# B&R Automation Studio project WRAPPER_CTRL
Automation Studio 4.9.6.42 SP; technology packages: mapp 1.63.0

## Configuration Errepi_P00936

CPU X20CP1301, AutomationRuntime O4.34, Build 4.1.2, Vc V4.72.7

### Task classes (Cpu.sw)
```
Cyclic#1 (cycle 8000 us, tolerance 8000 us):
  clock <- clock.prg
  Varie <- Varie.prg
  Program <- (binary)
Cyclic#2:
  main <- main.prg
Binaries: udbdef, TCData, sysconf, Role, User, iomap, ashwd, asfw, arconfig, ashwac
Libraries: FileIO, runtime, astime, asieccon, standard
```

### Hardware
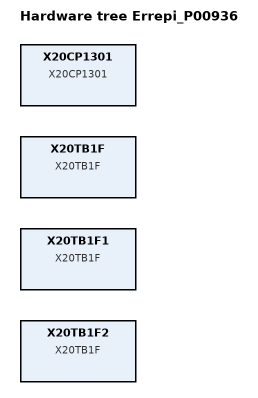
```
X20CP1301 : X20CP1301 v1.7.0.0  [X1 -> X1.SL; X2 -> X2.SL; X3 -> X3.SL]
  Module X1 (Type=X1, Virtual=true, Version=1.7.0.0)
    Connection (Connector=SS1, TargetModule=X20TB1F, TargetConnector=SS)
    Connection (Connector=SL, TargetModule=X20CP1301, TargetConnector=X1)
  Module X2 (Type=X2, Virtual=true, Version=1.7.0.0)
    Connection (Connector=SS1, TargetModule=X20TB1F1, TargetConnector=SS)
    Connection (Connector=SL, TargetModule=X20CP1301, TargetConnector=X2)
  Module X3 (Type=X3, Virtual=true, Version=1.7.0.0)
    Connection (Connector=SS1, TargetModule=X20TB1F2, TargetConnector=SS)
    Connection (Connector=SL, TargetModule=X20CP1301, TargetConnector=X3)
  Connector IF2:
    ActivateDevice = 1
    HostName = p00936
    Mode = Manual
    InternetAddress = 192.168.49.7
    SubnetMask = 255.255.255.0
    Vnc1
    VncVcObjectName1 = Visu
    VncKeyMappingFile1 = VC\PS2-Keyboard.dis
    VncAuthentication1 = 1
    VncPasswordViewOnly1 = errepi
    VncPasswordViewControl1 = promass
    ActivateSnmp = 2
  ConfigurationID = ERREPI_P00936
  ConfigVersion = 2022.5.1
  PermanentPvSize = 35
  RemanentGlobalPvSize = 45
  EnableUsbRemoteInstall = 1
  EnableCfRemoteInstall = 1
  RebootReset = 1
  Connections = 10
  TimerDeviceType = EPLX2X
  TimerDevice = X20CP1301.IF6
  TaskClassIdleTime = 8000
  Cyclic1Duration = 8000
  Cyclic1Tolerance = 8000
  Cyclic3Duration = 48000
  Cyclic3Tolerance = 48000
  Cyclic8Duration = 8000
  FileDevice1
  FileDeviceName1 = HD
  FileDevicePath1 = D:\RECIPES\
  FileDevice2
  FileDeviceName2 = CF
  FileDevicePath2 = D:\
  FileDevice3
  FileDeviceName3 = LOG
  FileDevicePath3 = D:\LOG\
  ActivateSntp = 1
  SntpcServAddr1 = 192.168.49.1
  SntpcServAddr2 = 8.8.8.8
  InternetFileSystemUsername = promass
  InternetFileSystemPassword = promass
  EthernetHostName = p00936
  EthernetDefaultGateway = 192.168.49.1
  FtpUser1
  FtpUsername1 = bazzica
  FtpUserPassword1 = fv7Wv821ewKqnMsDSvGQxxKgMMgXs+bZF/2FwIesLr0=  // promass
  FtpUserSalt1 = UDA6md8F
  FTPAccessRight1 = 0
  FTPMSPartition1 = DATA
  FtpUser2
  FtpUsername2 = errepi
  FtpUserPassword2 = knNz1PPTdcY0SkTRJpi6SMuvDsE3Y9gUDrG6vRz9RC4=  // errepi
  FtpUserSalt2 = Ww6eA1cq
  FTPAccessRight2 = 0
  FTPMSPartition2 = DATA
  ActivateOpcUa = 1
  OpcUaInformationModels_PV_Version = 1
X20TB1F : X20TB1F v1.0.0.0
X20TB1F1 : X20TB1F v1.0.0.0
X20TB1F2 : X20TB1F v1.0.0.0
```

### Cpu.per - X20CP1301/Cpu.per
```iecst
VAR_CONFIG
	gMac01LifeCounter AT %MD0; (* *)
	gMac01CounterOffset AT %MD4; (* *)
	gMac02LifeCounter AT %MD8; (* *)
	gMac02CounterOffset AT %MD12; (* *)
	gMac03LifeCounter AT %MD16; (* *)
	gMac03CounterOffset AT %MD20; (* *)
	glb_mac_name AT %M24; (* *)
END_VAR
```

## Configuration Errepi_P00987

CPU X20CP1301, AutomationRuntime O4.34, Build 4.1.2, Vc V4.72.7

### Hardware
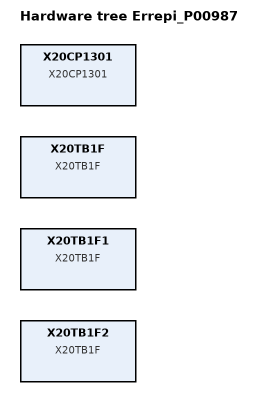
```
X20CP1301 : X20CP1301 v1.7.0.0  [X1 -> X1.SL; X2 -> X2.SL; X3 -> X3.SL]
  Module X1 (Type=X1, Virtual=true, Version=1.7.0.0)
    Connection (Connector=SS1, TargetModule=X20TB1F, TargetConnector=SS)
    Connection (Connector=SL, TargetModule=X20CP1301, TargetConnector=X1)
  Module X2 (Type=X2, Virtual=true, Version=1.7.0.0)
    Connection (Connector=SS1, TargetModule=X20TB1F1, TargetConnector=SS)
    Connection (Connector=SL, TargetModule=X20CP1301, TargetConnector=X2)
  Module X3 (Type=X3, Virtual=true, Version=1.7.0.0)
    Connection (Connector=SS1, TargetModule=X20TB1F2, TargetConnector=SS)
    Connection (Connector=SL, TargetModule=X20CP1301, TargetConnector=X3)
  Connector IF2:
    ActivateDevice = 1
    HostName = p00987
    Mode = Manual
    InternetAddress = 192.168.49.2
    SubnetMask = 255.255.255.0
    Vnc1
    VncVcObjectName1 = Visu
    VncKeyMappingFile1 = VC\PS2-Keyboard.dis
    VncAuthentication1 = 1
    VncPasswordViewOnly1 = errepi  // Password: errepi
    VncPasswordViewControl1 = promass  // Password: promass
    ActivateSnmp = 2
  ConfigurationID = ERREPI_P00987
  ConfigVersion = 2022.5.1
  PermanentPvSize = 35
  RemanentGlobalPvSize = 45
  EnableUsbRemoteInstall = 1
  EnableCfRemoteInstall = 1
  RebootReset = 1
  Connections = 10
  TimerDeviceType = EPLX2X
  TimerDevice = X20CP1301.IF6
  TaskClassIdleTime = 8000
  Cyclic1Duration = 8000
  Cyclic1Tolerance = 8000
  Cyclic3Duration = 48000
  Cyclic3Tolerance = 48000
  Cyclic8Duration = 8000
  FileDevice1
  FileDeviceName1 = HD
  FileDevicePath1 = D:\RECIPES\
  FileDevice2
  FileDeviceName2 = CF
  FileDevicePath2 = D:\
  FileDevice3
  FileDeviceName3 = LOG
  FileDevicePath3 = D:\LOG\
  ActivateSntp = 1
  SntpcServAddr1 = 192.168.49.1
  SntpcServAddr2 = 216.239.35.4
  InternetFileSystemUsername = promass
  InternetFileSystemPassword = promass
  EthernetHostName = p00987
  EthernetDefaultGateway = 192.168.49.1
  FtpUser1
  FtpUsername1 = bazzica
  FtpUserPassword1 = fv7Wv821ewKqnMsDSvGQxxKgMMgXs+bZF/2FwIesLr0=  // promass
  FtpUserSalt1 = UDA6md8F
  FTPAccessRight1 = 0
  FTPMSPartition1 = DATA
  FtpUser2
  FtpUsername2 = errepi
  FtpUserPassword2 = knNz1PPTdcY0SkTRJpi6SMuvDsE3Y9gUDrG6vRz9RC4=  // errepi
  FtpUserSalt2 = Ww6eA1cq
  FTPAccessRight2 = 0
  FTPMSPartition2 = DATA
  ActivateOpcUa = 1
  OpcUaInformationModels_PV_Version = 1
X20TB1F : X20TB1F v1.0.0.0
X20TB1F1 : X20TB1F v1.0.0.0
X20TB1F2 : X20TB1F v1.0.0.0
```

## Configuration SIM

CPU X20CP1382, AutomationRuntime D4.83, Build 4.1.2, Vc V4.72.7

### Hardware
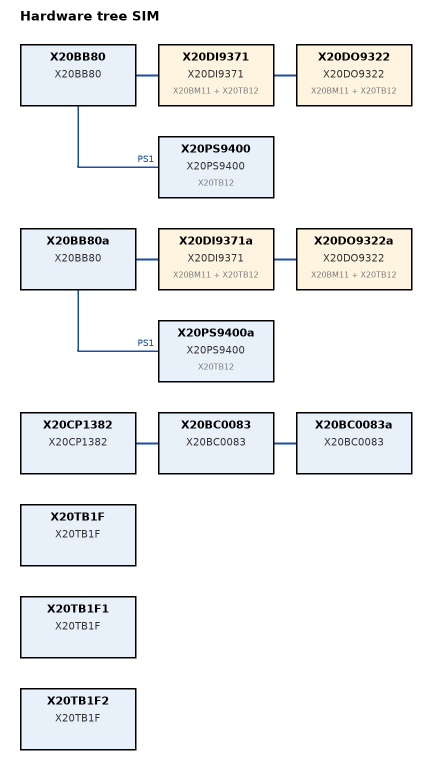
```
X20BB80 : X20BB80 v1.0.2.0
X20BB80a : X20BB80 v1.0.2.0
X20BC0083 : X20BC0083 v2.11.1.0  [PLK1 -> X20CP1382.IF3 (NodeNumber=1) [Cable Type=PowerlinkCable, Length=10, Version=1.0.0.3]; PLK2 -> X20BC0083a.PLK1 (NodeNumber=1) [Cable Type=PowerlinkCable, Length=10, Version=1.0.0.3]; SL -> X20BB80.SL1]
  Supervision = off
X20BC0083a : X20BC0083 v2.11.1.0  [PLK1 -> X20BC0083.PLK2 [Cable Type=PowerlinkCable, Length=10, Version=1.0.0.3]; SL -> X20BB80a.SL1]
  Supervision = off
X20BM11 : X20BM11 v1.0.0.1  [X2X1 -> X20BB80.IF1]
X20BM11a : X20BM11 v1.0.0.1  [X2X1 -> X20BB80a.IF1]
X20BM11b : X20BM11 v1.0.0.1  [X2X1 -> X20BM11.X2X2]
X20BM11c : X20BM11 v1.0.0.1  [X2X1 -> X20BM11a.X2X2]
X20CP1382 : X20CP1382 v1.11.0.0  [X1 -> X1.SL; X2 -> X2.SL; X3 -> X3.SL]
  Module X1 (Type=X1, Virtual=true, Version=1.11.0.0)
    Connection (Connector=SS1, TargetModule=X20TB1F, TargetConnector=SS)
    Connection (Connector=SL, TargetModule=X20CP1382, TargetConnector=X1)
  Module X2 (Type=X2, Virtual=true, Version=1.11.0.0)
    Connection (Connector=SS1, TargetModule=X20TB1F1, TargetConnector=SS)
    Connection (Connector=SL, TargetModule=X20CP1382, TargetConnector=X2)
  Module X3 (Type=X3, Virtual=true, Version=1.11.0.0)
    Connection (Connector=SS1, TargetModule=X20TB1F2, TargetConnector=SS)
    Connection (Connector=SL, TargetModule=X20CP1382, TargetConnector=X3)
  Connector IF2:
    ActivateDevice = 1
    HostName = promass
    Mode = Manual
    InternetAddress = 192.168.3.189  // TURQUEPLAST GIVEN IP
    SubnetMask = 255.255.255.0
    ActivateSnmp = 2
  Connector IF3:
    DNAConfiguration = manual
    CycleTime = 4000
  ConfigurationID = WRAPPER_CTRL_Turqueplast
  SimulationInaNodeNumber = 66
  PermanentPvSize = 1000
  RemanentGlobalPvSize = 20000
  EnableUsbRemoteInstall = 1
  EnableCfRemoteInstall = 1
  RebootReset = 1
  Connections = 10
  TimerDeviceType = EPLX2X
  TimerDevice = X20CP1382.IF3
  TaskClassIdleTime = 8000
  Cyclic1Duration = 8000
  Cyclic1Tolerance = 8000
  Cyclic3Duration = 48000
  Cyclic3Tolerance = 48000
  Cyclic8Duration = 8000
  FileDevice1
  FileDeviceName1 = HD
  FileDevicePath1 = C:\RECIPES\
  FileDevice2
  FileDeviceName2 = CF
  FileDevicePath2 = C:\
  FileDevice3
  FileDeviceName3 = LOG
  FileDevicePath3 = C:\LOG\
  EthernetHostName = promass
  EthernetDefaultGateway = 192.168.3.1
  FtpUser1
  FtpUsername1 = bazzica
  FtpUserPassword1 = VS/6Mr2ZWUxRpzYAgWdC7qPbhzWXz9kZH9v1k0AYU+w=
  FtpUserSalt1 = L4/axyh9
  FTPAccessRight1 = 0
  FTPdevice1 = ALL
  FtpUser2
  FtpUsername2 = turque
  FtpUserPassword2 = NA1x5qBXXFgCR/DJGfRfa8Sh4PrFzhFnpgUflhtmUyQ=
  FtpUserSalt2 = yY9t/zs3
  FTPdevice2 = ALL
X20DI9371 : X20DI9371 v1.1.0.0  [SS1 -> X20TB12b.SS; SL -> X20BM11.SL1]
  Supervision = off
X20DI9371a : X20DI9371 v1.1.0.0  [SS1 -> X20TB12c.SS; SL -> X20BM11a.SL1]
  Supervision = off
X20DO9322 : X20DO9322 v1.3.0.0  [SS1 -> X20TB12d.SS; SL -> X20BM11b.SL1]
  Supervision = off
X20DO9322a : X20DO9322 v1.3.0.0  [SS1 -> X20TB12e.SS; SL -> X20BM11c.SL1]
  Supervision = off
X20PS9400 : X20PS9400 v1.4.0.0  [SS1 -> X20TB12.SS; PS -> X20BB80.PS1]
  Supervision = off
X20PS9400a : X20PS9400 v1.4.0.0  [SS1 -> X20TB12a.SS; PS -> X20BB80a.PS1]
  Supervision = off
X20TB12 : X20TB12 v1.0.0.0
X20TB12a : X20TB12 v1.0.0.0
X20TB12b : X20TB12 v1.0.0.0
X20TB12c : X20TB12 v1.0.0.0
X20TB12d : X20TB12 v1.0.0.0
X20TB12e : X20TB12 v1.0.0.0
X20TB1F : X20TB1F v1.0.0.0
X20TB1F1 : X20TB1F v1.0.0.0
X20TB1F2 : X20TB1F v1.0.0.0
```

### IoMap.iom - X20CP1382/IoMap.iom
```iecst
VAR_CONFIG
	::gPWL02_ok AT %IX."X20BC0083a".ModuleOk;
	::gPWL01_ok AT %IX."X20BC0083".ModuleOk;
END_VAR
```

## Configuration Turqueplast

CPU X20CP1382, AutomationRuntime D4.83, Build 4.1.2, Vc V4.72.7

### Task classes (Cpu.sw)
```
Cyclic#1 (cycle 8000 us, tolerance 8000 us):
  clock <- LOGIC.clock.prg
  Varie <- VARIOUS.Varie.prg
  Program <- (binary)
Cyclic#2:
  main <- LOGIC.main.prg
Binaries: udbdef, TCData, sysconf, Role, User, iomap, ashwd, asfw, arconfig, ashwac
Libraries: FileIO, runtime, astime, asieccon, standard
```

### Hardware
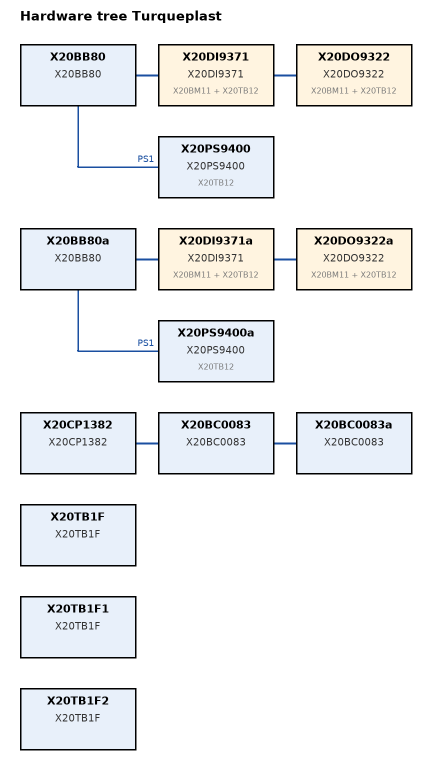
```
X20BB80 : X20BB80 v1.0.2.0
X20BB80a : X20BB80 v1.0.2.0
X20BC0083 : X20BC0083 v2.11.1.0  [PLK1 -> X20CP1382.IF3 (NodeNumber=1) [Cable Type=PowerlinkCable, Length=10, Version=1.0.0.3]; PLK2 -> X20BC0083a.PLK1 (NodeNumber=1) [Cable Type=PowerlinkCable, Length=10, Version=1.0.0.3]; SL -> X20BB80.SL1]
  Supervision = off
X20BC0083a : X20BC0083 v2.11.1.0  [PLK1 -> X20BC0083.PLK2 [Cable Type=PowerlinkCable, Length=10, Version=1.0.0.3]; SL -> X20BB80a.SL1]
  Supervision = off
X20BM11 : X20BM11 v1.0.0.1  [X2X1 -> X20BB80.IF1]
X20BM11a : X20BM11 v1.0.0.1  [X2X1 -> X20BB80a.IF1]
X20BM11b : X20BM11 v1.0.0.1  [X2X1 -> X20BM11.X2X2]
X20BM11c : X20BM11 v1.0.0.1  [X2X1 -> X20BM11a.X2X2]
X20CP1382 : X20CP1382 v1.11.0.0  [X1 -> X1.SL; X2 -> X2.SL; X3 -> X3.SL]
  Module X1 (Type=X1, Virtual=true, Version=1.11.0.0)
    Connection (Connector=SS1, TargetModule=X20TB1F, TargetConnector=SS)
    Connection (Connector=SL, TargetModule=X20CP1382, TargetConnector=X1)
  Module X2 (Type=X2, Virtual=true, Version=1.11.0.0)
    Connection (Connector=SS1, TargetModule=X20TB1F1, TargetConnector=SS)
    Connection (Connector=SL, TargetModule=X20CP1382, TargetConnector=X2)
  Module X3 (Type=X3, Virtual=true, Version=1.11.0.0)
    Connection (Connector=SS1, TargetModule=X20TB1F2, TargetConnector=SS)
    Connection (Connector=SL, TargetModule=X20CP1382, TargetConnector=X3)
  Connector IF2:
    ActivateDevice = 1
    HostName = promass
    Mode = Manual
    InternetAddress = 192.168.3.189  // TURQUEPLAST GIVEN IP
    SubnetMask = 255.255.255.0
    ActivateSnmp = 2
  Connector IF3:
    DNAConfiguration = manual
    CycleTime = 4000
  ConfigurationID = WRAPPER_CTRL_Turqueplast
  Simulation = 1
  SimulationInaNodeNumber = 66
  PermanentPvSize = 1000
  RemanentGlobalPvSize = 20000
  EnableUsbRemoteInstall = 1
  EnableCfRemoteInstall = 1
  RebootReset = 1
  Connections = 10
  TimerDeviceType = EPLX2X
  TimerDevice = X20CP1382.IF3
  TaskClassIdleTime = 8000
  Cyclic1Duration = 8000
  Cyclic1Tolerance = 8000
  Cyclic3Duration = 48000
  Cyclic3Tolerance = 48000
  Cyclic8Duration = 8000
  FileDevice1
  FileDeviceName1 = HD
  FileDevicePath1 = C:\RECIPES\
  FileDevice2
  FileDeviceName2 = CF
  FileDevicePath2 = C:\
  FileDevice3
  FileDeviceName3 = LOG
  FileDevicePath3 = C:\LOG\
  EthernetHostName = promass
  EthernetDefaultGateway = 192.168.3.1
  FtpUser1
  FtpUsername1 = bazzica
  FtpUserPassword1 = VS/6Mr2ZWUxRpzYAgWdC7qPbhzWXz9kZH9v1k0AYU+w=
  FtpUserSalt1 = L4/axyh9
  FTPAccessRight1 = 0
  FTPdevice1 = ALL
  FtpUser2
  FtpUsername2 = turque
  FtpUserPassword2 = NA1x5qBXXFgCR/DJGfRfa8Sh4PrFzhFnpgUflhtmUyQ=
  FtpUserSalt2 = yY9t/zs3
  FTPdevice2 = ALL
X20DI9371 : X20DI9371 v1.1.0.0  [SS1 -> X20TB12b.SS; SL -> X20BM11.SL1]
  Supervision = off
X20DI9371a : X20DI9371 v1.1.0.0  [SS1 -> X20TB12c.SS; SL -> X20BM11a.SL1]
  Supervision = off
X20DO9322 : X20DO9322 v1.3.0.0  [SS1 -> X20TB12d.SS; SL -> X20BM11b.SL1]
  Supervision = off
X20DO9322a : X20DO9322 v1.3.0.0  [SS1 -> X20TB12e.SS; SL -> X20BM11c.SL1]
  Supervision = off
X20PS9400 : X20PS9400 v1.4.0.0  [SS1 -> X20TB12.SS; PS -> X20BB80.PS1]
  Supervision = off
X20PS9400a : X20PS9400 v1.4.0.0  [SS1 -> X20TB12a.SS; PS -> X20BB80a.PS1]
  Supervision = off
X20TB12 : X20TB12 v1.0.0.0
X20TB12a : X20TB12 v1.0.0.0
X20TB12b : X20TB12 v1.0.0.0
X20TB12c : X20TB12 v1.0.0.0
X20TB12d : X20TB12 v1.0.0.0
X20TB12e : X20TB12 v1.0.0.0
X20TB1F : X20TB1F v1.0.0.0
X20TB1F1 : X20TB1F v1.0.0.0
X20TB1F2 : X20TB1F v1.0.0.0
```

### IoMap.iom - X20CP1382/IoMap.iom
```iecst
VAR_CONFIG
	gMAC03raw.Di.Run AT %IX."X2".DigitalInput01;
	gMAC03raw.Di.Alarm AT %IX."X2".DigitalInput02;
	gMAC03raw.Di.MoldChange AT %IX."X2".DigitalInput03;
	gMAC03raw.Di.Manual AT %IX."X2".DigitalInput04;
	gMAC03raw.Di.NewCycleSignal AT %IX."X2".DigitalInput05;
	gMAC03raw.Di.CommitEnd AT %IX."X2".DigitalInput06;
	gMAC02raw.Di.Run AT %IX."X20DI9371".DigitalInput01;
	gMAC02raw.Di.Alarm AT %IX."X20DI9371".DigitalInput02;
	gMAC02raw.Di.MoldChange AT %IX."X20DI9371".DigitalInput03;
	gMAC02raw.Di.Manual AT %IX."X20DI9371".DigitalInput04;
	gMAC02raw.Di.NewCycleSignal AT %IX."X20DI9371".DigitalInput05;
	gMAC02raw.Di.CommitEnd AT %IX."X20DI9371".DigitalInput06;
	gMAC01raw.Di.Run AT %IX."X20DI9371a".DigitalInput01;
	gMAC01raw.Di.Alarm AT %IX."X20DI9371a".DigitalInput02;
	gMAC01raw.Di.MoldChange AT %IX."X20DI9371a".DigitalInput03;
	gMAC01raw.Di.Manual AT %IX."X20DI9371a".DigitalInput04;
	gMAC01raw.Di.NewCycleSignal AT %IX."X20DI9371a".DigitalInput05;
	gMAC01raw.Di.CommitEnd AT %IX."X20DI9371a".DigitalInput06;
	::gPWL02_ok AT %IX."X20BC0083a".ModuleOk;
	::gPWL01_ok AT %IX."X20BC0083".ModuleOk;
	gPWL03_ok AT %IX."X2".DigitalInput07;
	::glbMac02On AT %IX."X20DI9371".DigitalInput07;
	::glbMac01On AT %IX."X20DI9371a".DigitalInput07;
END_VAR
```

## Logical view

Binary libraries used (declarations not repeated): operator, runtime, astime, AsIecCon, FileIO, standard, asstring

### Global.var - Global variables
```iecst
VAR
	M3_NewCycle : TON;
	M2_NewCycle : TON;
	M1_NewCycle : TON;
	M1_AUTO_1s : TON;
	gPWL03_ok : BOOL;
	gPWL02_ok : BOOL;
	gPWL01_ok : BOOL;
	gPulse_500 : BOOL;
	gPulse_100 : BOOL;
	gMAC03raw : typIO;
END_VAR
VAR RETAIN
	gMac03LifeCounter : DINT;
	gMac03CounterOffset : DINT;
END_VAR
VAR
	gMAC03 : {REDUND_UNREPLICABLE} typOmronMachine := (0);
	gMAC02raw : typIO;
END_VAR
VAR RETAIN
	gMac02LifeCounter : DINT;
	gMac02CounterOffset : DINT;
END_VAR
VAR
	gMAC02 : {REDUND_UNREPLICABLE} typOmronMachine := (0);
	gMAC01raw : typIO;
END_VAR
VAR RETAIN
	gMac01LifeCounter : DINT;
	gMac01CounterOffset : DINT;
END_VAR
VAR
	gMAC01 : {REDUND_UNREPLICABLE} typOmronMachine := (0);
	glbMac02On : BOOL;
	glbMac01On : BOOL;
END_VAR
VAR RETAIN
	glbClock : tGlbClock;
END_VAR
VAR
	gCounter03 : BOOL;
	gCounter02 : BOOL;
	gCounter01 : BOOL;
	g1secTick01 : BOOL;
	cpu_time_start_mac03 : UDINT;
	cpu_time_start_mac02 : UDINT;
	cpu_time_start_mac01 : UDINT;
	cmdClock : tCmdClock;
END_VAR
VAR RETAIN
	glb_mac_name : STRING[10];
END_VAR
```


### Program Logical/LOGIC/main (IEC)

#### Cyclic.ld
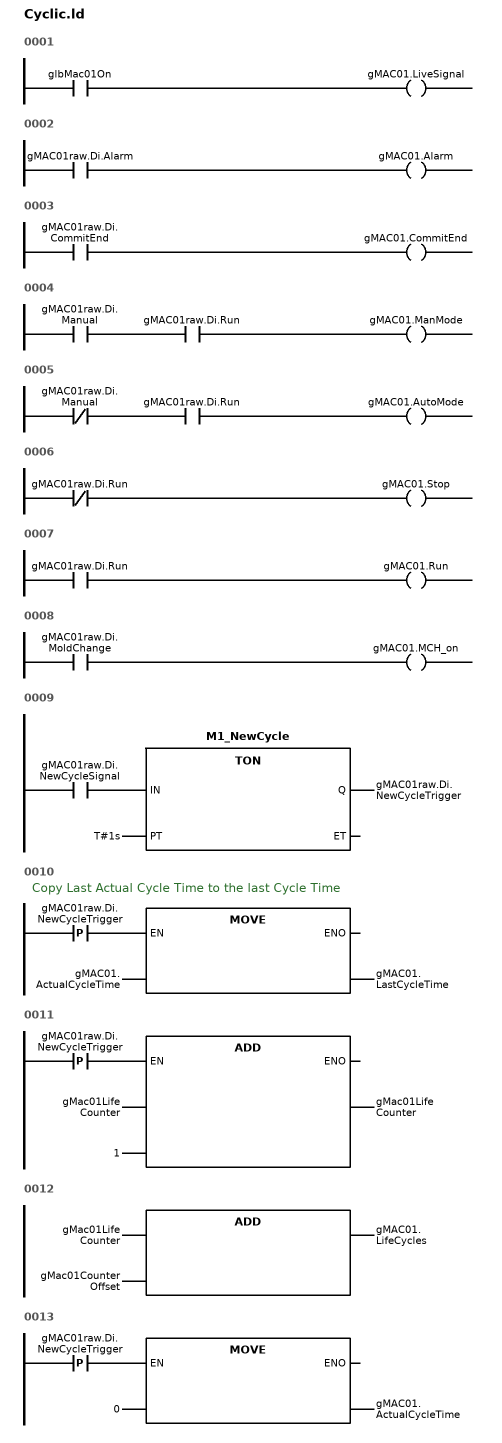
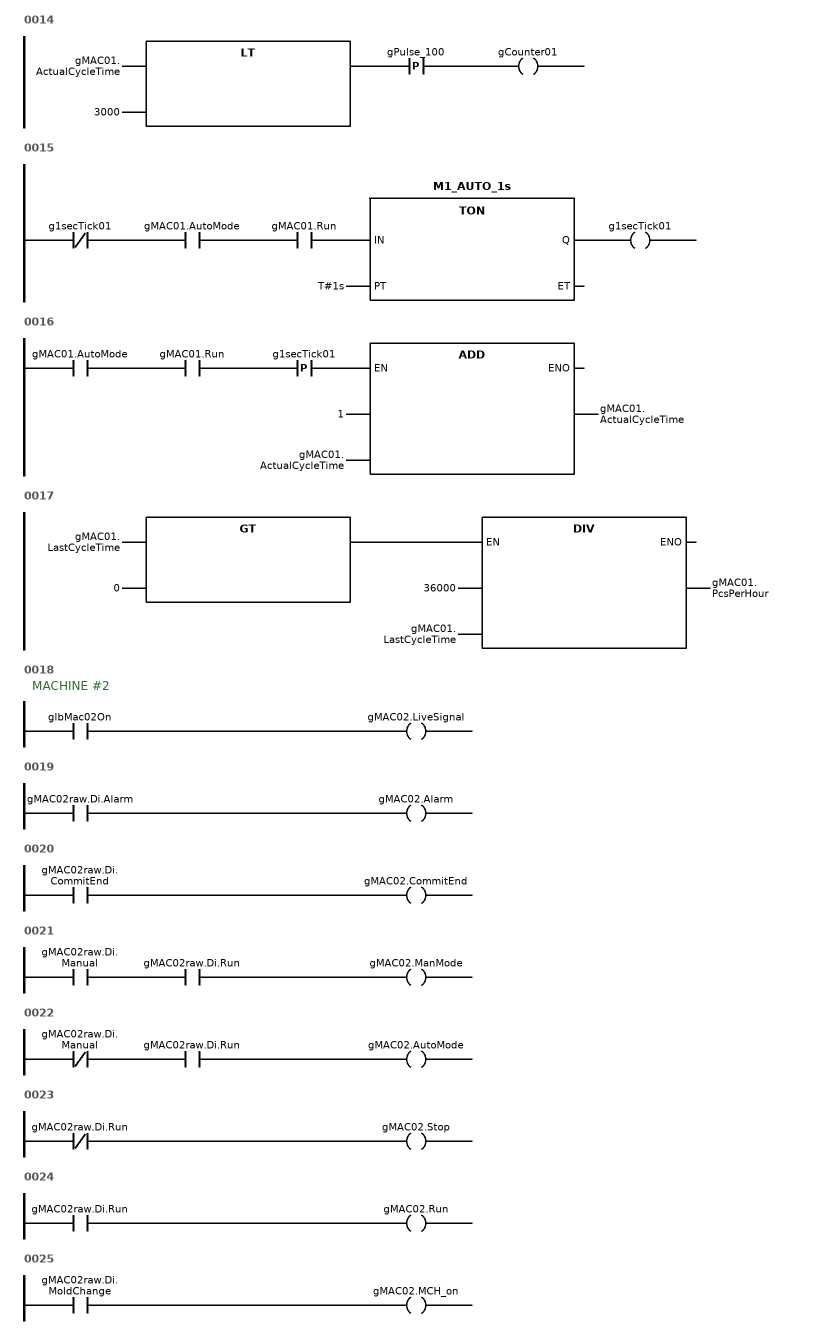
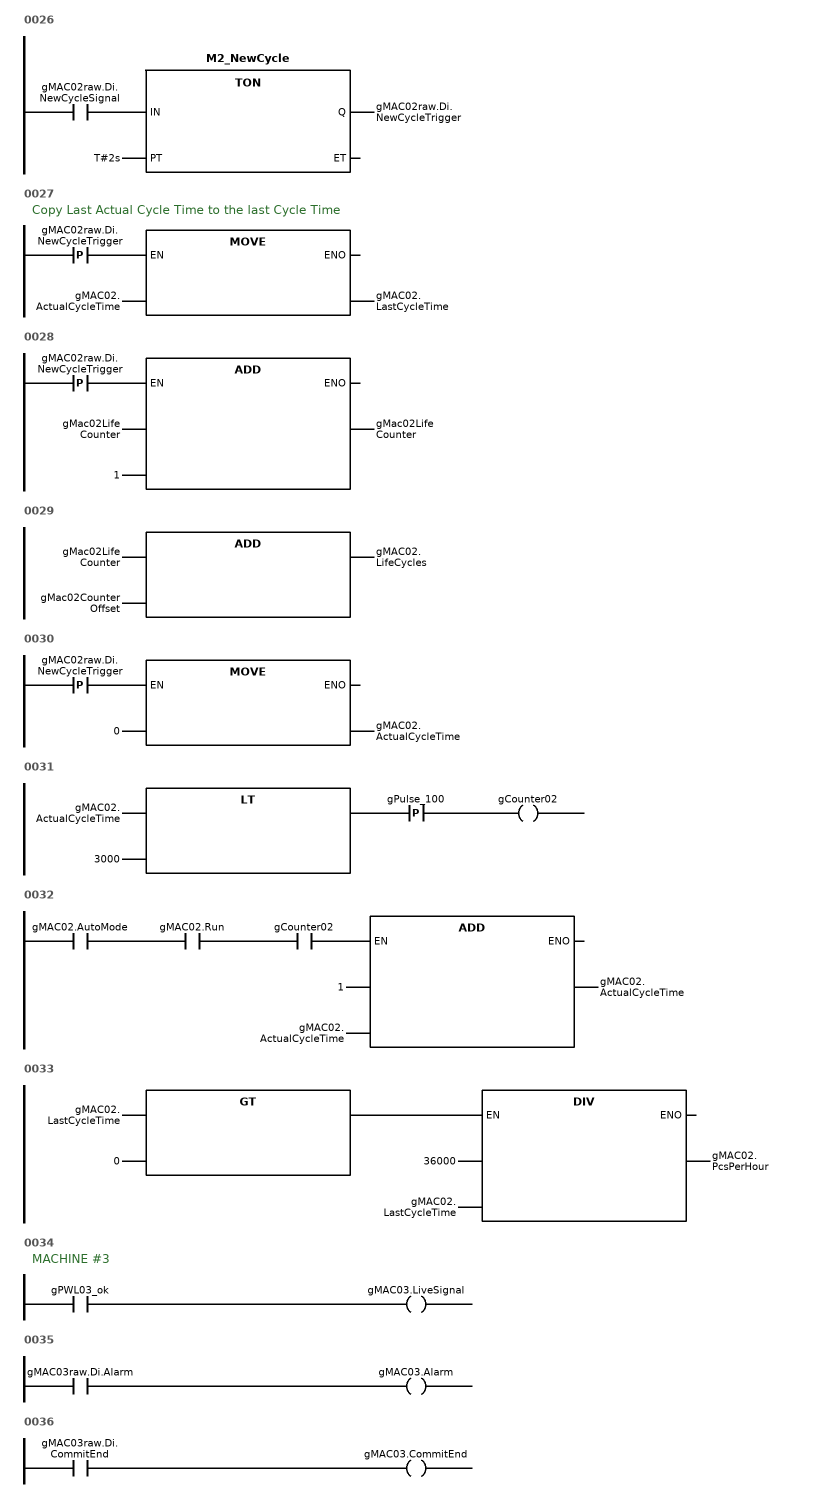
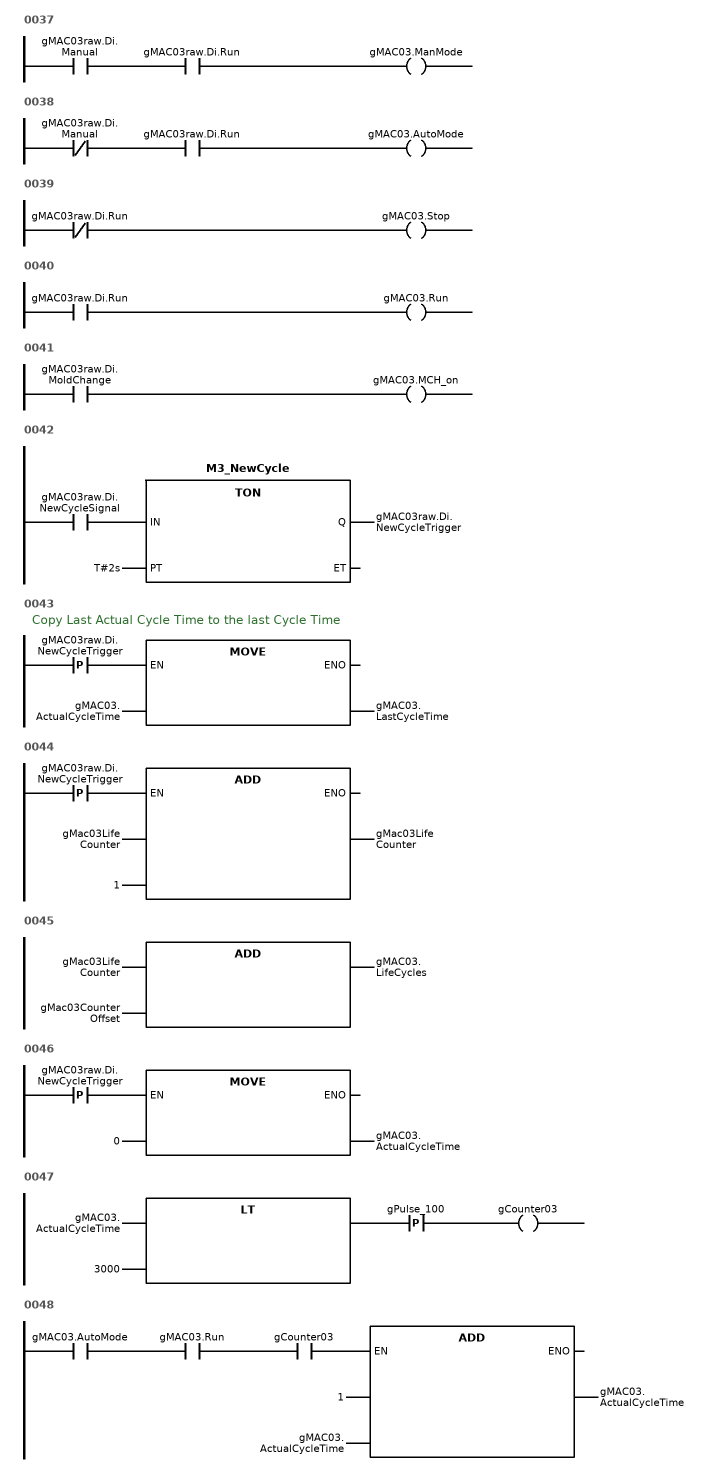
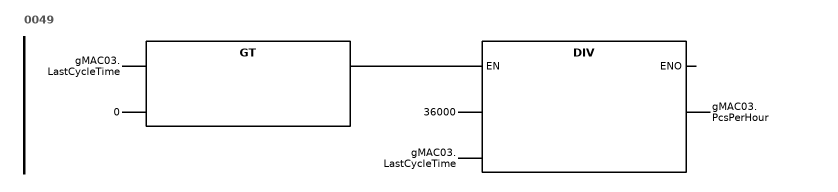
Ladder, written as Structured Text:
```iecst
PROGRAM _CYCLIC
VAR
    _e1 : R_TRIG;
    _e2 : R_TRIG;
    _e3 : R_TRIG;
    _e4 : R_TRIG;
    _e5 : R_TRIG;
    _p6 : BOOL;
    _p7 : BOOL;
    _e8 : R_TRIG;
    _e9 : R_TRIG;
    _e10 : R_TRIG;
    _e11 : R_TRIG;
    _p12 : BOOL;
    _p13 : BOOL;
    _e14 : R_TRIG;
    _e15 : R_TRIG;
    _e16 : R_TRIG;
    _e17 : R_TRIG;
    _p18 : BOOL;
    _p19 : BOOL;
END_VAR
(* Network 1 *)
gMAC01.LiveSignal := glbMac01On;

(* Network 2 *)
gMAC01.Alarm := gMAC01raw.Di.Alarm;

(* Network 3 *)
gMAC01.CommitEnd := gMAC01raw.Di.CommitEnd;

(* Network 4 *)
gMAC01.ManMode := gMAC01raw.Di.Manual AND gMAC01raw.Di.Run;

(* Network 5 *)
gMAC01.AutoMode := NOT gMAC01raw.Di.Manual AND gMAC01raw.Di.Run;

(* Network 6 *)
gMAC01.Stop := NOT gMAC01raw.Di.Run;

(* Network 7 *)
gMAC01.Run := gMAC01raw.Di.Run;

(* Network 8 *)
gMAC01.MCH_on := gMAC01raw.Di.MoldChange;

(* Network 9 *)
M1_NewCycle(IN := gMAC01raw.Di.NewCycleSignal, PT := T#1s);
gMAC01raw.Di.NewCycleTrigger := M1_NewCycle.Q;

(* Network 10: Copy Last Actual Cycle Time to the last Cycle Time *)
_e1(CLK := gMAC01raw.Di.NewCycleTrigger);
IF _e1.Q THEN gMAC01.LastCycleTime := gMAC01.ActualCycleTime; END_IF;

(* Network 11 *)
_e2(CLK := gMAC01raw.Di.NewCycleTrigger);
IF _e2.Q THEN gMac01LifeCounter := gMac01LifeCounter + 1; END_IF;

(* Network 12 *)
gMAC01.LifeCycles := gMac01LifeCounter + gMac01CounterOffset;

(* Network 13 *)
_e3(CLK := gMAC01raw.Di.NewCycleTrigger);
IF _e3.Q THEN gMAC01.ActualCycleTime := 0; END_IF;

(* Network 14 *)
_e4(CLK := gPulse_100);
gCounter01 := (gMAC01.ActualCycleTime < 3000) AND _e4.Q;

(* Network 15 *)
M1_AUTO_1s(IN := NOT g1secTick01 AND gMAC01.AutoMode AND gMAC01.Run, PT := T#1s);
g1secTick01 := M1_AUTO_1s.Q;

(* Network 16 *)
_e5(CLK := g1secTick01);
_p6 := gMAC01.AutoMode AND gMAC01.Run AND _e5.Q;
IF _p6 THEN gMAC01.ActualCycleTime := 1 + gMAC01.ActualCycleTime; END_IF;

(* Network 17 *)
_p7 := gMAC01.LastCycleTime > 0;
IF _p7 THEN gMAC01.PcsPerHour := 36000 / gMAC01.LastCycleTime; END_IF;

(* Network 18: MACHINE #2 *)
gMAC02.LiveSignal := glbMac02On;

(* Network 19 *)
gMAC02.Alarm := gMAC02raw.Di.Alarm;

(* Network 20 *)
gMAC02.CommitEnd := gMAC02raw.Di.CommitEnd;

(* Network 21 *)
gMAC02.ManMode := gMAC02raw.Di.Manual AND gMAC02raw.Di.Run;

(* Network 22 *)
gMAC02.AutoMode := NOT gMAC02raw.Di.Manual AND gMAC02raw.Di.Run;

(* Network 23 *)
gMAC02.Stop := NOT gMAC02raw.Di.Run;

(* Network 24 *)
gMAC02.Run := gMAC02raw.Di.Run;

(* Network 25 *)
gMAC02.MCH_on := gMAC02raw.Di.MoldChange;

(* Network 26 *)
M2_NewCycle(IN := gMAC02raw.Di.NewCycleSignal, PT := T#2s);
gMAC02raw.Di.NewCycleTrigger := M2_NewCycle.Q;

(* Network 27: Copy Last Actual Cycle Time to the last Cycle Time *)
_e8(CLK := gMAC02raw.Di.NewCycleTrigger);
IF _e8.Q THEN gMAC02.LastCycleTime := gMAC02.ActualCycleTime; END_IF;

(* Network 28 *)
_e9(CLK := gMAC02raw.Di.NewCycleTrigger);
IF _e9.Q THEN gMac02LifeCounter := gMac02LifeCounter + 1; END_IF;

(* Network 29 *)
gMAC02.LifeCycles := gMac02LifeCounter + gMac02CounterOffset;

(* Network 30 *)
_e10(CLK := gMAC02raw.Di.NewCycleTrigger);
IF _e10.Q THEN gMAC02.ActualCycleTime := 0; END_IF;

(* Network 31 *)
_e11(CLK := gPulse_100);
gCounter02 := (gMAC02.ActualCycleTime < 3000) AND _e11.Q;

(* Network 32 *)
_p12 := gMAC02.AutoMode AND gMAC02.Run AND gCounter02;
IF _p12 THEN gMAC02.ActualCycleTime := 1 + gMAC02.ActualCycleTime; END_IF;

(* Network 33 *)
_p13 := gMAC02.LastCycleTime > 0;
IF _p13 THEN gMAC02.PcsPerHour := 36000 / gMAC02.LastCycleTime; END_IF;

(* Network 34: MACHINE #3 *)
gMAC03.LiveSignal := gPWL03_ok;

(* Network 35 *)
gMAC03.Alarm := gMAC03raw.Di.Alarm;

(* Network 36 *)
gMAC03.CommitEnd := gMAC03raw.Di.CommitEnd;

(* Network 37 *)
gMAC03.ManMode := gMAC03raw.Di.Manual AND gMAC03raw.Di.Run;

(* Network 38 *)
gMAC03.AutoMode := NOT gMAC03raw.Di.Manual AND gMAC03raw.Di.Run;

(* Network 39 *)
gMAC03.Stop := NOT gMAC03raw.Di.Run;

(* Network 40 *)
gMAC03.Run := gMAC03raw.Di.Run;

(* Network 41 *)
gMAC03.MCH_on := gMAC03raw.Di.MoldChange;

(* Network 42 *)
M3_NewCycle(IN := gMAC03raw.Di.NewCycleSignal, PT := T#2s);
gMAC03raw.Di.NewCycleTrigger := M3_NewCycle.Q;

(* Network 43: Copy Last Actual Cycle Time to the last Cycle Time *)
_e14(CLK := gMAC03raw.Di.NewCycleTrigger);
IF _e14.Q THEN gMAC03.LastCycleTime := gMAC03.ActualCycleTime; END_IF;

(* Network 44 *)
_e15(CLK := gMAC03raw.Di.NewCycleTrigger);
IF _e15.Q THEN gMac03LifeCounter := gMac03LifeCounter + 1; END_IF;

(* Network 45 *)
gMAC03.LifeCycles := gMac03LifeCounter + gMac03CounterOffset;

(* Network 46 *)
_e16(CLK := gMAC03raw.Di.NewCycleTrigger);
IF _e16.Q THEN gMAC03.ActualCycleTime := 0; END_IF;

(* Network 47 *)
_e17(CLK := gPulse_100);
gCounter03 := (gMAC03.ActualCycleTime < 3000) AND _e17.Q;

(* Network 48 *)
_p18 := gMAC03.AutoMode AND gMAC03.Run AND gCounter03;
IF _p18 THEN gMAC03.ActualCycleTime := 1 + gMAC03.ActualCycleTime; END_IF;

(* Network 49 *)
_p19 := gMAC03.LastCycleTime > 0;
IF _p19 THEN gMAC03.PcsPerHour := 36000 / gMAC03.LastCycleTime; END_IF;
END_PROGRAM
```

#### Init.ld
Ladder, written as Structured Text:
```iecst
PROGRAM _INIT
END_PROGRAM
```

### Program Logical/LOGIC/clock (ANSIC, version 0.00.0)

- Visualisation Logical/HMI/Visu (not shown)

### Program Logical/VARIOUS/Varie (ANSIC)

#### Variables.var
```iecst
VAR
	pulse_100_start_time : UDINT;
	pulse_500_start_time : UDINT;
	pulse_750_start_time : UDINT;
END_VAR
```

#### Cyclic.c
```c
#include <bur/plctypes.h>

#ifdef _DEFAULT_INCLUDES
	#include <AsDefault.h>
#endif

void _CYCLIC ProgramCyclic(void)
{
	// Genero una variabile pulse da 500ms
	if ((glbClock.cpu_time - pulse_500_start_time > 250) && !gPulse_500)
	{
		pulse_500_start_time 	= glbClock.cpu_time;
		gPulse_500  = 1;
	}
	else if ((glbClock.cpu_time - pulse_500_start_time > 250) && gPulse_500)
	{
		pulse_500_start_time 	= glbClock.cpu_time;
		gPulse_500  = 0;
	}

	// Genero una variabile pulse da 100ms
	if ((glbClock.cpu_time - pulse_100_start_time > 50) && !gPulse_100)
	{
		pulse_100_start_time 	= glbClock.cpu_time;
		gPulse_100  = 1;
	}
	else if ((glbClock.cpu_time - pulse_100_start_time > 50) && gPulse_100)
	{
		pulse_100_start_time 	= glbClock.cpu_time;
		gPulse_100  = 0;
	}

}
```

### Program Logical/VARIOUS/OpcUA_IF (IEC)

#### Types.typ
```iecst
TYPE
	typMacStatus : 	STRUCT
		stop : BOOL;
		man : BOOL;
		running : BOOL;
		auto : BOOL;
		alarm : BOOL;
		mch_on : BOOL;
		commit_cycles : UDINT;
		actual_cycle_nr : UDINT;
		last_cycle_time : UDINT;
		actual_cycle_time : UDINT;
	END_STRUCT;
END_TYPE
```

#### Variables.var
```iecst
VAR
	life_cycles : REFERENCE TO UDINT;
	life_mold_distance : REFERENCE TO LREAL; (*Distanza totale in metri*)
	mac_status : typMacStatus;
END_VAR
```

#### Cyclic.st
```iecst
	PROGRAM _CYCLIC
	(* Insert code here *)

//	life_cycles	UDINT	TRUE	FALSE	FALSE	FALSE		 	 	 	2
//	life_mold_distance	LREAL	FALSE	FALSE	FALSE	TRUE		Distanza totale in metri			3
//	life_auto_mode_wrk_time	typ_work_time	FALSE	FALSE	FALSE	TRUE		 	 	 	4
//	life_loading_1_total_wrk_time	typ_work_time	FALSE	FALSE	FALSE	TRUE		 	 	 	5
//	life_loading_2_total_wrk_time	typ_work_time	FALSE	FALSE	FALSE	TRUE		 	 	 	6
//	life_hydraulic_total_wrk_time	typ_work_time	FALSE	FALSE	FALSE	TRUE		 	 	 	7
//	life_manu_mode_wrk_time	typ_work_time	FALSE	FALSE	FALSE	TRUE		 	 	 	8
//	life_total_wrk_time	typ_work_time	FALSE	FALSE	FALSE	TRUE		 	 	 	9
//	recipe	typ_Recipe	TRUE	FALSE	FALSE	FALSE		 	 	 	10
//	last_recipe	STRING[30]	TRUE	FALSE	FALSE	FALSE	 	 	 	 	11
//	life_total_mold_change	USINT	FALSE	FALSE	FALSE	TRUE		 	 	 	12
//	power_analyzer	typ_Ctr_Master_memory	FALSE	FALSE	FALSE	TRUE		 	 	 	13
//	mac_status	typMacStatus	FALSE	FALSE	FALSE	TRUE	 	 	 	 	14

	//glb_remote_recipe_loading				:= 1;		// used to enable popup and relative

	life_cycles ACCESS ADR(gMAC01.LifeCycles);

	//power_analyzer ACCESS ADR(machine.Ctr_MPaster_data.memory);
	//mac_status ACCESS ADR(permanent_ore_auto);

	mac_status.actual_cycle_nr		:= gMAC01.ActualCycleNr;
	mac_status.actual_cycle_time	:= gMAC01.ActualCycleTime;
	//mac_status.commit_cycles		:=
	mac_status.last_cycle_time		:= gMAC01.LastCycleTime;
	mac_status.auto					:= gMAC01.AutoMode;
	mac_status.man					:= gMAC01.ManMode;
	mac_status.alarm				:= gMAC01.Alarm;
	mac_status.stop					:= gMAC01.Stop;
	mac_status.running				:= gMAC01.Run;
	mac_status.mch_on				:= gMAC01.MCH_on;

END_PROGRAM
```

#### Init.st
```iecst
PROGRAM _INIT
	(* Insert code here *)
//	glb_rem_recipe_load_cmd	:=0; strcmp(ADR(glb_mac_name), ADR("P00987")) = 0)
	IF (strcmp(ADR(glb_mac_name), ADR("P00987")) = 0) THEN
		;
	ELSE
		;
	END_IF;

END_PROGRAM
```

### Program Logical/clock

#### clock.var
```iecst
VAR
	ulCheckRam	:UDINT;
	locClock	:tLocClock;
	dataGetTime	:DTGetTime;
	dataSetTime	:DTSetTime;
END_VAR
```

#### clock.c
```c
#ifdef _DEFAULT_INCLUDES
 #include <AsDefault.h>
#endif
/*=============================================================================
                      			PROMASS S.r.l.
=============================================================================*/

/******************************************************************************
    INCLUSIONE HEADER FILES
******************************************************************************/

#include <bur\plctypes.h>
#include <string.h>
#include <AsTime.h>  /* libreria 'AsTime' */

/******************************************************************************
    SIMBOLI
******************************************************************************/

#define CHECK_RAM_CODE    0xA7FF252C     /* per la verifica di validità ram */

/******************************************************************************
    STRUTTURE E TIPI LOCALI (UTILIZZATI SOLO IN QUESTO FILE)
******************************************************************************/

/******************************************************************************
    PROTOTIPI DELLE FUNZIONI AUSILIARIE (DEFINITE IN QUESTO FILE)
******************************************************************************/

/******************************************************************************
    VARIABILI _GLOBAL (AUTOMATION STUDIO)
******************************************************************************/

/******************************************************************************
    VARIABILI _LOCAL (AUTOMATION STUDIO)
******************************************************************************/

/******************************************************************************
    VARIABILI GLOBALI (C ANSI)
******************************************************************************/

/******************************************************************************
    MACRO
******************************************************************************/

/******************************************************************************
    FUNZIONE DI INIZIALIZZAZIONE DELLA TASK
******************************************************************************/

void _INIT TaskInit(void)
{
	/* Azzera sempre le _GLOBAL prodotte in questa task */
	memset(&glbClock, 0, sizeof(glbClock));
	memset(&cmdClock, 0, sizeof(cmdClock));

	/* Verifica la validità della RAM dati */
	if(ulCheckRam != CHECK_RAM_CODE)            /* RAM non valida? */
	{
		/* Azzera le _LOCAL ritentive */
		memset(&locClock, 0, sizeof(locClock));

		/* Registra allarme */
		glbClock.alRamData = 1;

		/* Assegna il codice di validazione RAM */
		ulCheckRam = CHECK_RAM_CODE;
	}

	/* Registra l'orario di spegnimento */
	locClock.rtcShutDown = locClock.rtcRuntime; /* leggo il valore dal dato runtime in memoria */

	if(locClock.rtcShutDown == 0) /* Orario errato? */
	{
		/* Sì: registra l'allarme */
		 glbClock.alRtcShutDown = 1;
	}

	/* Richiesta dell'orario di accensione */
	dataGetTime.enable = 1;
	DTGetTime(&dataGetTime);

	if(dataGetTime.status == 0) /* L'orario di sistema è valido? */
	{
		/* Sì: registra l'orario ottenuto */
		locClock.rtcStartUp = dataGetTime.DT1;

	}
	else
	{
		/* No: registra il valore nullo */
		locClock.rtcStartUp = 0;

		/* Registra allarme */
		glbClock.alRtcStartUp = 1;
	}

	/* Calcolo del tempo di spegnimento [secondi] */
	if( (locClock.rtcStartUp != 0)&&(locClock.rtcShutDown != 0) ) /* Orari di accensione e spegnimento validi? */
	{
		/* Sì: calcola il tempo di spegnimento */
		locClock.ulTimePlcOff =  DiffDT(locClock.rtcStartUp, locClock.rtcShutDown);
	}
	else
	{
		/* No: assegna valore nullo */
		locClock.ulTimePlcOff = 0;
	}

	/* Tempo di spegnimento global */
	if( (locClock.ulTimePlcOff != 0)                           &&  /* E' stato possibile calcolare il tempo di spegnimento? */
		(locClock.ulTimePlcOff != 0xFFFFFFFF)                  )   /* Il tempo di spegnimento è sensato (non negativo)?     */
	{
		glbClock.ulTimePlcOff = locClock.ulTimePlcOff;
	}
	else
	{
		glbClock.ulTimePlcOff = 0;
	}

	/* Orari di accensione e spegnimento in forma 'Calendar' (_GLOBAL)  */

	if(locClock.rtcStartUp != 0) /* orario accensione valido? */
	{
		/* Sì: convertilo in 'Calendar' */
		DT_TO_DTStructure(locClock.rtcStartUp, (unsigned long)&glbClock.calStartUp);
	}
	else
	{
		/* No: azzera la struttura 'Calendar' */
		memset((void*)&glbClock.calStartUp, 0, sizeof(glbClock.calStartUp));
	}

	if(locClock.rtcShutDown != 0) /* orario spegnimento valido? */
	{
		/* Sì: convertilo in 'Calendar' */
		DT_TO_DTStructure(locClock.rtcShutDown, (unsigned long)&glbClock.calShutDown);
	}
	else
	{
		/* No: azzera la struttura 'Calendar' */
		memset((void*)&glbClock.calShutDown, 0, sizeof(glbClock.calShutDown));
	}

} /* fine _INIT */

/******************************************************************************
   FUNZIONE CICLICA DELLA TASK
******************************************************************************/

void _CYCLIC TaskCyclic(void)
{

	/*===== RILIEVO COMANDO DI SETTAGGIO "REAL TIME CLOCK" =====*/

	if(cmdClock.bSetClock) /* E' stato richiesto il settaggio? */
	{
		/* azzera i flag  di risposta */
		cmdClock.bOkSet    = 0;
        cmdClock.bErSet    = 0;

        /* converti l'orario in forma 'date time' */
		locClock.rtcSetTime = DTStructure_TO_DT((UDINT) &cmdClock.calSetTime);

		/* richiedi il settaggio del RealTimeClock*/
		dataSetTime.enable = 1;
		dataSetTime.DT1    = locClock.rtcSetTime;
		DTSetTime(&dataSetTime);

		/* verifica l'esito del settaggio e definisci il flag di risposta */
		if(dataSetTime.status == 0)   cmdClock.bOkSet = 1; /* esito positivo */
  		else                          cmdClock.bErSet = 1; /* esito negativo */

  		/* Annulla il comando */
		cmdClock.bSetClock = 0;
	}

	/*===== RILIEVO ORARIO ATTUALE =====*/

	dataGetTime.enable = 1;
	DTGetTime(&dataGetTime);

	if(dataGetTime.status == 0) /* L'orario di sistema è valido? */
	{
		/* Sì: registra l'orario ottenuto */
		locClock.rtcRuntime = dataGetTime.DT1;

	}
	else
	{
		/* No: assegna il valore nullo */
		locClock.rtcRuntime = 0;

		/* Registra l'allarme */
		glbClock.alRtcRuntime = 1;
	}

	/* Orario _GLOBAL */
	glbClock.rtcRuntime = locClock.rtcRuntime;

	/*===== TEMPO DALLO STARTUP [msec] =====*/

	locClock.myTime      = clock_ms(); /* _LOCAL */
	glbClock.cpu_time    = (UDINT)locClock.myTime;

} /* fine _CYCLIC */

/******************************************************************************
   DEFINIZIONE DELLE FUNZIONI AUSILIARIE
******************************************************************************/
```

### Program Logical/main

#### Exit.ld
Ladder, written as Structured Text:
```iecst
PROGRAM _EXIT
END_PROGRAM
```

Listed in the project but not available here: Logical/Global.typ, Logical/LOGIC/clock/clock.var, Logical/LOGIC/clock/clock.c, Logical/CFG
